Universal Robots PolyScope program: Servoj_rtde_example.urp

Program Servoj_rtde_example (installation=default directory=/programs/RemoteOperation createdIn=3.2.19275.0 lastSavedIn=5.10.0.106268 robotSerialNumber=20185500191)
Calibrated DH parameters: a=[0.000131, -0.165639, -0.102041, 0.000082, 0.000046, 0]; d=[0.162455, 220.258006, 1988.136334, -2208.260978, 0.099826, 0.099896]; alpha=[1.570482, -0.001777, -0.000172, 1.570393, -1.570735, 0]; deltaTheta=[0, -1.170526, -0.137148, 1.307669, -0.000001, 0]
BeforeStart
  Script: write_output_boolean_register(0,  True )
  Wait Sleep waitTime=0.01
  mode := 0
  j := [0.,0,0,0,0,0]
Robot Program (runOnlyOnce=true)
  Script: write_output_boolean_register(0,  False )
  Script: mode = read_input_integer_register(0)
  Loop While (checkContinuously=false) expression=mode < 3
    Loop While (checkContinuously=false) expression=mode ≟ 1
      MoveJ speed 15 deg/s, acceleration 40 deg/s^2 (useActiveTCP=true) feature=Base
        Waypoint Waypoint (Variable): variable(name=j)
      Script: write_output_boolean_register(0, True )
      Script: mode = read_input_integer_register(0)
      Script: sync()
    Loop While (checkContinuously=false) expression=(mode ≟ 2)
      SuppressedNode
        Script: servoj(j, lookahead_time=0.05, gain=3000)
      Script: servoj(j)
      Script: mode = read_input_integer_register(0)
    Script: mode = read_input_integer_register(0)
    Script: sync()
Thread Thread_1 (runOnlyOnce=false)
  Loop Forever
    tmp := [0,0,0,0,0,0]
    Script: tmp[0] = read_input_float_register(0)
    Script: tmp[1] = read_input_float_register(1)
    Script: tmp[2] = read_input_float_register(2)
    Script: tmp[3] = read_input_float_register(3)
    Script: tmp[4] = read_input_float_register(4)
    Script: tmp[5] = read_input_float_register(5)
    j := tmp
    Script: sync()
